FUNCTION_BLOCK SM_QuantityValue
VAR_INPUT
	///Numeric value
	{attribute 'OPC.UA.DA' := '1'}
	{attribute 'OPC.UA.DA.Access' := '1'}
	value: LREAL;
	///Unit of the numeric value
	{attribute 'OPC.UA.DA' := '1'}
	{attribute 'OPC.UA.DA.Access' := '1'}
	unit: Units;
END_VAR
VAR_OUTPUT
	///Current status description
	{attribute 'OPC.UA.DA' := '1'}
	{attribute 'OPC.UA.DA.Access' := '1'}
	actualStatus: STRING;
END_VAR
VAR_IN_OUT
END_VAR
VAR
END_VAR

END_FUNCTION_BLOCK

(* stored: Version 1.1.0.1, ProductVersion 3.1.4019.2
   POU SM_QuantityValue: Id {40a7928d-c724-4ccf-8f22-a4bc8f886de5}, SpecialFunc None *)
